FUNCTION_BLOCK fbCylinderCtrl

VAR_INPUT
	IN_CylName:STRING;
	In_Enable:BOOL;
	In_Reset:BOOL;
	(*Sensors*)
	In_WorkRS:BOOL;
	In_HomeRS:BOOL;	
	(*Timer*)
	In_WorkTON:TIME;
	In_HomeTON:TIME;
	in_Timeout:TIME;
END_VAR

VAR_OUTPUT
	Out_WorkSV:BOOL;
	Out_HomeSV:BOOL;	
END_VAR

VAR_IN_OUT
	CylVar:structCylinder;
	Station:structStationCtrl;
END_VAR

VAR

	Loc_Work:BOOL;
	Loc_Home:BOOL;
	Err_Cyl:BOOL;
	Fwd_TOut: TON;
	Bwd_TOut: TON;
	Fwd_TON: TON;
	Bwd_TON: TON;
	Loc_WorkPls: BOOL;
	FwdPls: R_TRIG;
	BwdPls: R_TRIG;
	Loc_HomePls: BOOL;
	Out_RSErr:BOOL;
	FwdPosPls: F_TRIG;
	BwdPosPls: F_TRIG;
END_VAR
VAR // added by the converter: edge detectors and wires of the graphical bodies
    _w1, _w2, _w3, _w4, _w5 : BOOL;
END_VAR

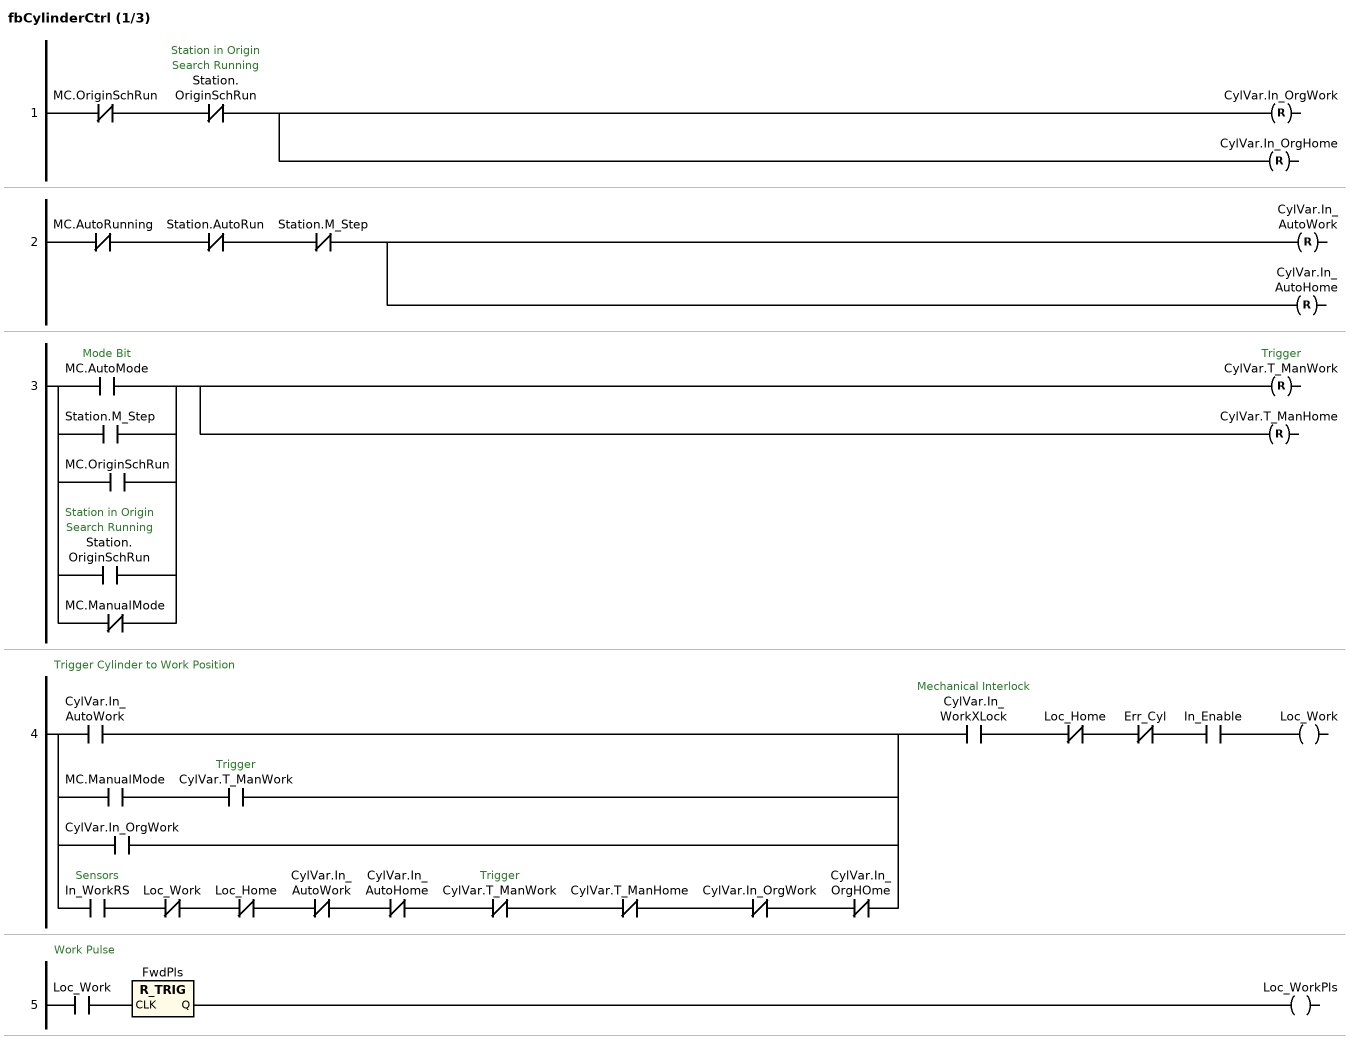
// NETWORK 1
//   Station.OriginSchRun: Station in Origin Search Running
_w1 := NOT MC.OriginSchRun AND NOT Station.OriginSchRun;
CylVar.In_OrgWork R= _w1;
CylVar.In_OrgHome R= _w1;

// NETWORK 2
_w2 := NOT MC.AutoRunning AND NOT Station.AutoRun AND NOT Station.M_Step;
CylVar.In_AutoWork R= _w2;
CylVar.In_AutoHome R= _w2;

// NETWORK 3
//   MC.AutoMode: Mode Bit
//   Station.OriginSchRun: Station in Origin Search Running
//   CylVar.T_ManWork: Trigger
_w3 := MC.AutoMode OR Station.M_Step OR MC.OriginSchRun OR Station.OriginSchRun OR NOT MC.ManualMode;
CylVar.T_ManWork R= _w3;
CylVar.T_ManHome R= _w3;

// NETWORK 4
// Trigger Cylinder to Work Position
//   CylVar.T_ManWork: Trigger
//   In_WorkRS: Sensors
//   CylVar.In_WorkXLock: Mechanical Interlock
Loc_Work := (CylVar.In_AutoWork OR MC.ManualMode AND CylVar.T_ManWork OR CylVar.In_OrgWork OR In_WorkRS AND NOT Loc_Work AND NOT Loc_Home AND NOT CylVar.In_AutoWork AND NOT CylVar.In_AutoHome AND NOT CylVar.T_ManWork AND NOT CylVar.T_ManHome AND NOT CylVar.In_OrgWork AND NOT CylVar.In_OrgHOme) AND CylVar.In_WorkXLock AND NOT Loc_Home AND NOT Err_Cyl AND In_Enable;

// NETWORK 5
// Work Pulse
FwdPls(CLK := Loc_Work); // R_TRIG
Loc_WorkPls := FwdPls.Q;

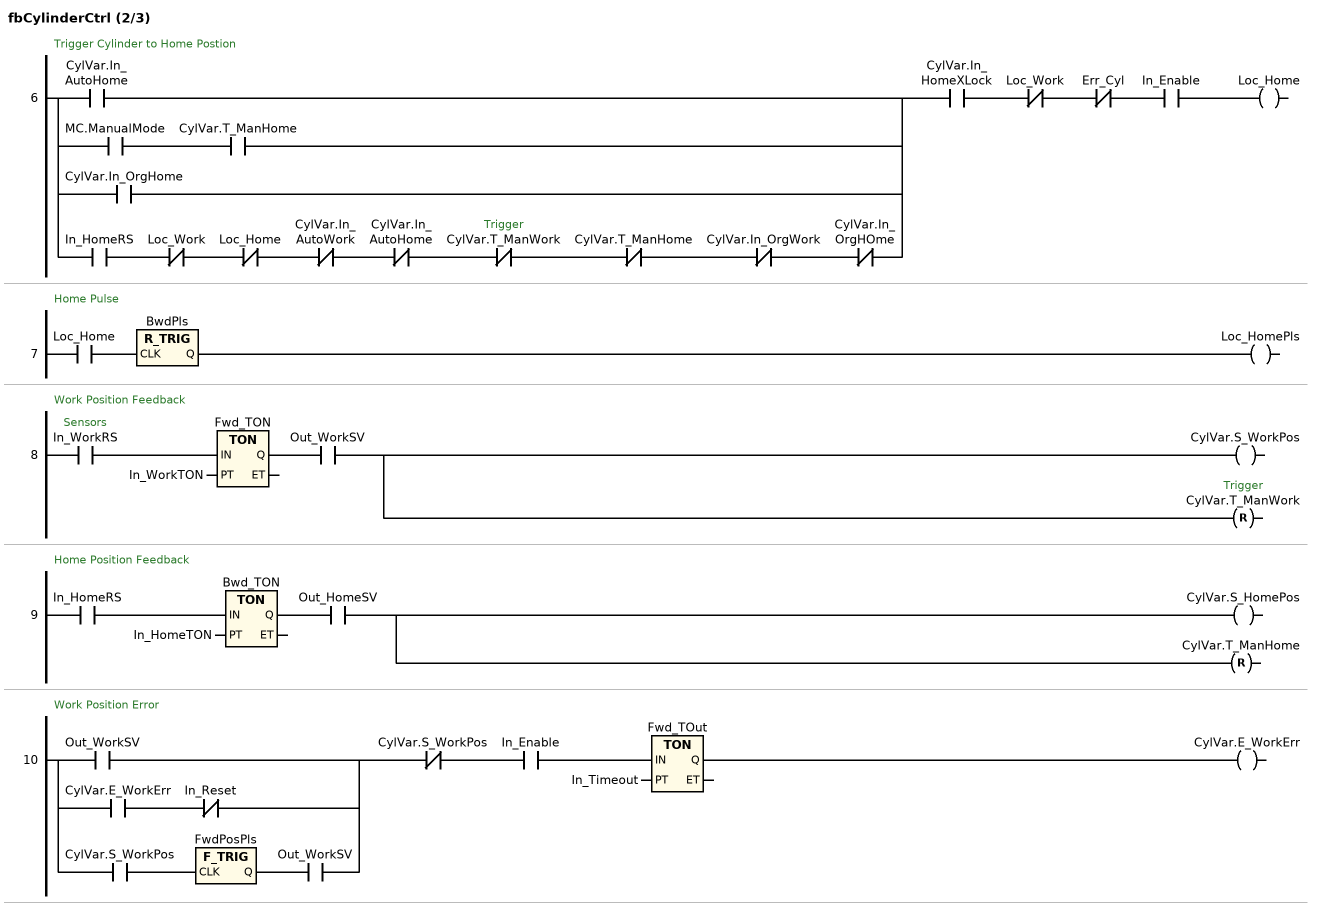
// NETWORK 6
// Trigger Cylinder to Home Postion
//   CylVar.T_ManWork: Trigger
Loc_Home := (CylVar.In_AutoHome OR MC.ManualMode AND CylVar.T_ManHome OR CylVar.In_OrgHome OR In_HomeRS AND NOT Loc_Work AND NOT Loc_Home AND NOT CylVar.In_AutoWork AND NOT CylVar.In_AutoHome AND NOT CylVar.T_ManWork AND NOT CylVar.T_ManHome AND NOT CylVar.In_OrgWork AND NOT CylVar.In_OrgHOme) AND CylVar.In_HomeXLock AND NOT Loc_Work AND NOT Err_Cyl AND In_Enable;

// NETWORK 7
// Home Pulse
BwdPls(CLK := Loc_Home); // R_TRIG
Loc_HomePls := BwdPls.Q;

// NETWORK 8
// Work Position Feedback
//   In_WorkRS: Sensors
//   In_WorkTON: Timer
//   CylVar.T_ManWork: Trigger
Fwd_TON(IN := In_WorkRS, PT := In_WorkTON); // TON
_w4 := Fwd_TON.Q AND Out_WorkSV;
CylVar.S_WorkPos := _w4;
CylVar.T_ManWork R= _w4;

// NETWORK 9
// Home Position Feedback
Bwd_TON(IN := In_HomeRS, PT := In_HomeTON); // TON
_w5 := Bwd_TON.Q AND Out_HomeSV;
CylVar.S_HomePos := _w5;
CylVar.T_ManHome R= _w5;

// NETWORK 10
// Work Position Error
FwdPosPls(CLK := CylVar.S_WorkPos); // F_TRIG
Fwd_TOut(IN := (Out_WorkSV OR CylVar.E_WorkErr AND NOT In_Reset OR FwdPosPls.Q AND Out_WorkSV) AND NOT CylVar.S_WorkPos AND In_Enable, PT := In_Timeout); // TON
CylVar.E_WorkErr := Fwd_TOut.Q;

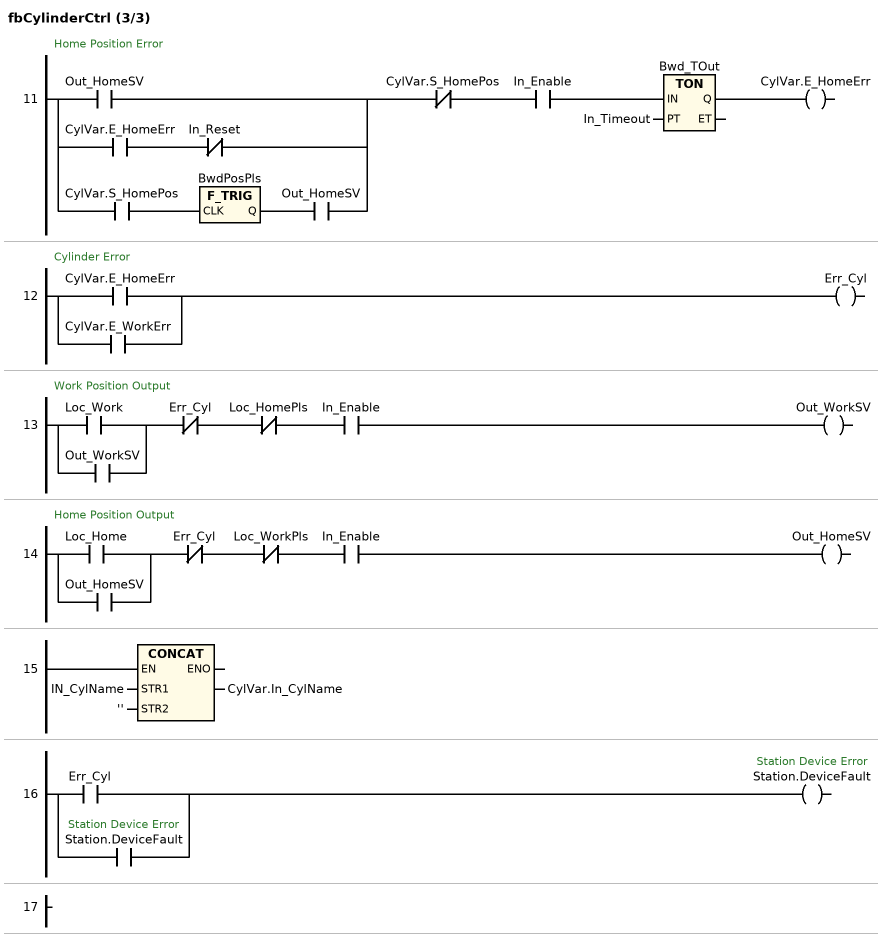
// NETWORK 11
// Home Position Error
BwdPosPls(CLK := CylVar.S_HomePos); // F_TRIG
Bwd_TOut(IN := (Out_HomeSV OR CylVar.E_HomeErr AND NOT In_Reset OR BwdPosPls.Q AND Out_HomeSV) AND NOT CylVar.S_HomePos AND In_Enable, PT := In_Timeout); // TON
CylVar.E_HomeErr := Bwd_TOut.Q;

// NETWORK 12
// Cylinder Error
Err_Cyl := CylVar.E_HomeErr OR CylVar.E_WorkErr;

// NETWORK 13
// Work Position Output
Out_WorkSV := (Loc_Work OR Out_WorkSV) AND NOT Err_Cyl AND NOT Loc_HomePls AND In_Enable;

// NETWORK 14
// Home Position Output
Out_HomeSV := (Loc_Home OR Out_HomeSV) AND NOT Err_Cyl AND NOT Loc_WorkPls AND In_Enable;

// NETWORK 15
CylVar.In_CylName := CONCAT(STR1 := IN_CylName, STR2 := '');

// NETWORK 16
//   Station.DeviceFault: Station Device Error
Station.DeviceFault := Err_Cyl OR Station.DeviceFault;

// NETWORK 17

END_FUNCTION_BLOCK

(* stored: Version 1.1.0.1, ProductVersion 3.1.4018.2
   POU fbCylinderCtrl: Id {66c52f80-8d81-4cda-8e6b-ea36dcddef2d}, SpecialFunc None *)
